FUNCTION_BLOCK DigitalOutput EXTENDS BaseIO
VAR_INPUT
	Value: BOOL;
	Override: BOOL;
	OverrideValue: BOOL;
END_VAR
VAR_OUTPUT
	ProcessValue: BOOL;
	OffTime: LTIME;
	OnTime: LTIME;
END_VAR
VAR
	InitDone: BOOL;
	TempValue: BOOL;
	TimeChange: LTIME;
	LastValue: BOOL;
END_VAR
VAR PERSISTENT
	Inverted: BOOL;
	SavedOverride: BOOL;
	SavedOverrideValue: BOOL;
END_VAR

SUPER^();
IF NOT InitDone THEN
	InitDone := TRUE;
	OverrideValue := SavedOverrideValue;
	Override := SavedOverride;	
	TimeChange := LTIME();
END_IF
SavedOverride := Override;
SavedOverrideValue := OverrideValue;

IF NOT Override THEN
	TempValue := Value;
ELSE
	TempValue := OverrideValue;	
END_IF

IF Inverted THEN
	TempValue := NOT TempValue;
END_IF

ProcessValue := TempValue;

IF ProcessValue <> LastValue THEN
	LastValue := ProcessValue;
	TimeChange := LTIME();
END_IF

IF NOT ProcessValue THEN
	OffTime := LTIME() - TimeChange;
ELSE
	OffTime := LTIME#0S;
END_IF

IF ProcessValue THEN
	OnTime := LTIME() - TimeChange;
ELSE
	OnTime := LTIME#0s;
END_IF

END_FUNCTION_BLOCK

(* stored: Version 1.1.0.1, ProductVersion 3.1.4024.4
   POU DigitalOutput: Id {46b6ab89-acfc-4cfb-91a5-2ccc6ebe02db}, SpecialFunc None *)
